(* Logix 5000 project; controller BreakGroup_US vendor 1 type 14 code 211 rev 32.16; software revision 32.05; part 6 of 8 *)
(* tags used below, declared in another part *)
   Emg_Stop : BOOL;
   HMI_ACK : BOOL;
   HMI_MAN_STN_120_STOP : BOOL;
   HMI_MAN_STN_30_STOP : BOOL;
   HMI_MAN_STN_40_STOP : BOOL;
   HMI_STN30_GRI_SETPOINT : REAL;
   HMI_STN30_HORIZ_MOVE_SETPOINT : REAL;
   HMI_STN30_VER_LIFTUP_SETPOINT : REAL;
   HMI_STN30_VER_PICK_SETPOINT : REAL;
   HMI_STN40_GRI_GRIP_POINT : REAL;
   HMI_STN40_GRI_SETPOINT : REAL;
   HMI_STN40_HORIZ_MOVE_SETPOINT : REAL;
   HMI_STN40_VER_LIFTUP_SETPOINT : REAL;
   HMI_STN40_VER_PICK_LIFTUP_SETPOINT : REAL;
   HMI_STN40_VER_PICK_SETPOINT : REAL;
   HMI_STN40_VER_PLACE_SETPOINT : REAL;
   MAN_STN_120_HOME : TIMER;
   MAN_STN_30_HOME : TIMER;
   MAN_STN_40_HOME : TIMER;
   MCP_GY_01_Gripper : MCP_Servo_01;
   MCP_GY_01_Horizontal : MCP_Servo_02;
   MCP_GY_01_Vertical : MCP_Servo_02;
   MCP_ST_30_Turntable_Motor : MCP_Servo_02;
   MCP_ST_40_Turntable_Motor : MCP_Servo_02;
   RCP_ST_120_Turntable_Motor : RCP_Servo_02;
   ST10_Trolley1Lock_Cyl_01_Extended : ALIAS FOR MCP_PT01:1:I.0;
   ST_120_Start : BOOL;
   ST_30_Start : BOOL;
   ST_40_Start : BOOL;
   STN_120_Connection_fault : BOOL;
   STN_120_Conveyor : INDEX_Block;
   STN_120_HMI_PB : SINT[2];
   STN_30_Auto_ENable : BOOL;
   STN_30_HMI_PB : SINT;
   STN_30_PRE_COND_OK : BOOL;
   STN_30_SEQ : DINT;
   STN_30_SEQUENCE_AUTO : SINT;
   STN_40_HMI_PB : SINT;
   STN_40_PRE_COND_OK : BOOL;
   STN_40_SEQ : DINT;
   STN_40_SEQUENCE_AUTO : SINT;
   T10_01 : TIMER;
   T11_01 : TIMER;
   T1_01 : TIMER;
   T2_01 : TIMER;
   T3_01 : TIMER;
   T4_01 : TIMER;
   T5_01 : TIMER;
   T6_01 : TIMER;
   T7_01 : TIMER;
   T8_01 : TIMER;
   T9_01 : TIMER;
   Test_COND_OK : DINT;
(* Station_120, continued *)

ROUTINE Manual   (* ladder *)
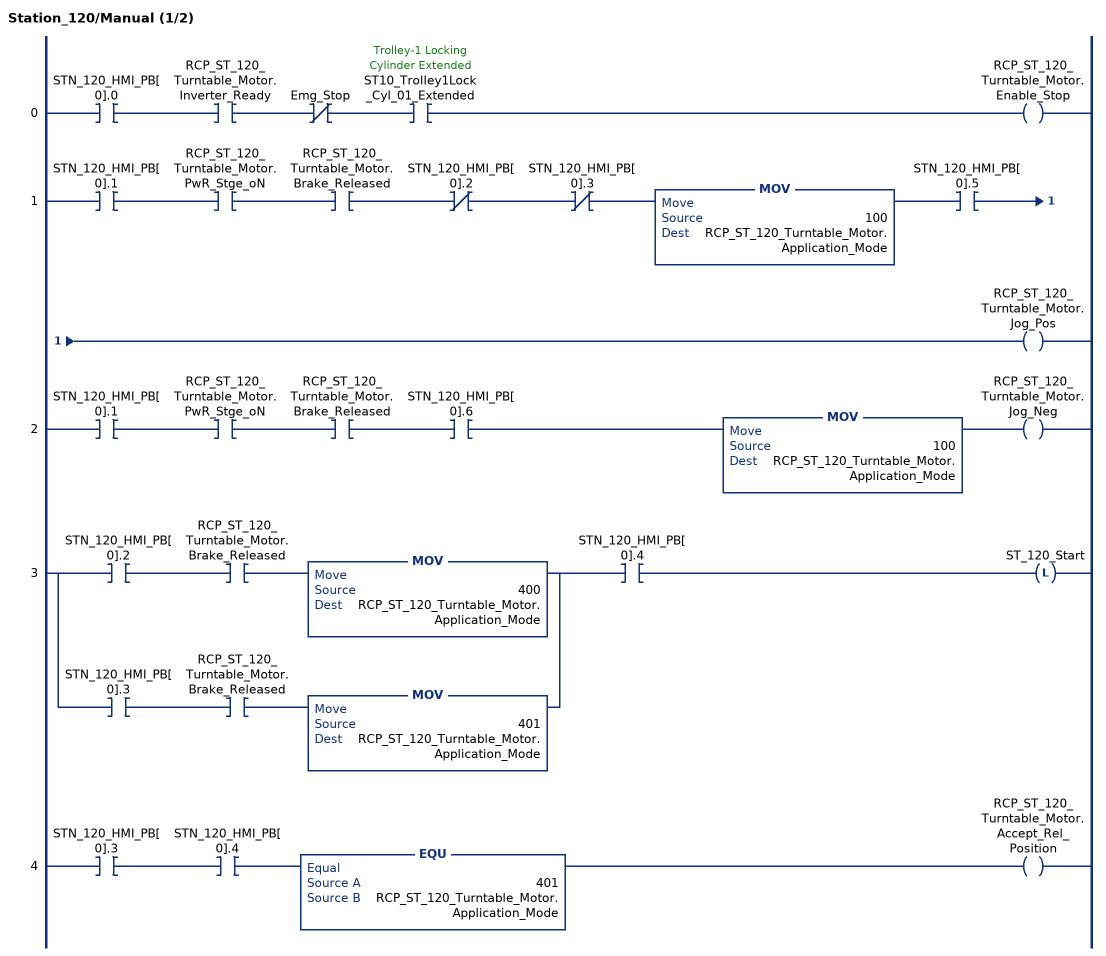
   0: XIC(STN_120_HMI_PB[0].0)XIC(RCP_ST_120_Turntable_Motor.Inverter_Ready)XIO(Emg_Stop)XIC(ST10_Trolley1Lock_Cyl_01_Extended)OTE(RCP_ST_120_Turntable_Motor.Enable_Stop);
   1: XIC(STN_120_HMI_PB[0].1)XIC(RCP_ST_120_Turntable_Motor.PwR_Stge_oN)XIC(RCP_ST_120_Turntable_Motor.Brake_Released)XIO(STN_120_HMI_PB[0].2)XIO(STN_120_HMI_PB[0].3)MOV(100,RCP_ST_120_Turntable_Motor.Application_Mode)XIC(STN_120_HMI_PB[0].5)OTE(RCP_ST_120_Turntable_Motor.Jog_Pos);
   2: XIC(STN_120_HMI_PB[0].1)XIC(RCP_ST_120_Turntable_Motor.PwR_Stge_oN)XIC(RCP_ST_120_Turntable_Motor.Brake_Released)XIC(STN_120_HMI_PB[0].6)MOV(100,RCP_ST_120_Turntable_Motor.Application_Mode)OTE(RCP_ST_120_Turntable_Motor.Jog_Neg);
   3: [XIC(STN_120_HMI_PB[0].2) XIC(RCP_ST_120_Turntable_Motor.Brake_Released) MOV(400,RCP_ST_120_Turntable_Motor.Application_Mode) ,XIC(STN_120_HMI_PB[0].3) XIC(RCP_ST_120_Turntable_Motor.Brake_Released) MOV(401,RCP_ST_120_Turntable_Motor.Application_Mode) ]XIC(STN_120_HMI_PB[0].4)OTL(ST_120_Start);
   4: XIC(STN_120_HMI_PB[0].3)XIC(STN_120_HMI_PB[0].4)EQU(401,RCP_ST_120_Turntable_Motor.Application_Mode)OTE(RCP_ST_120_Turntable_Motor.Accept_Rel_Position);
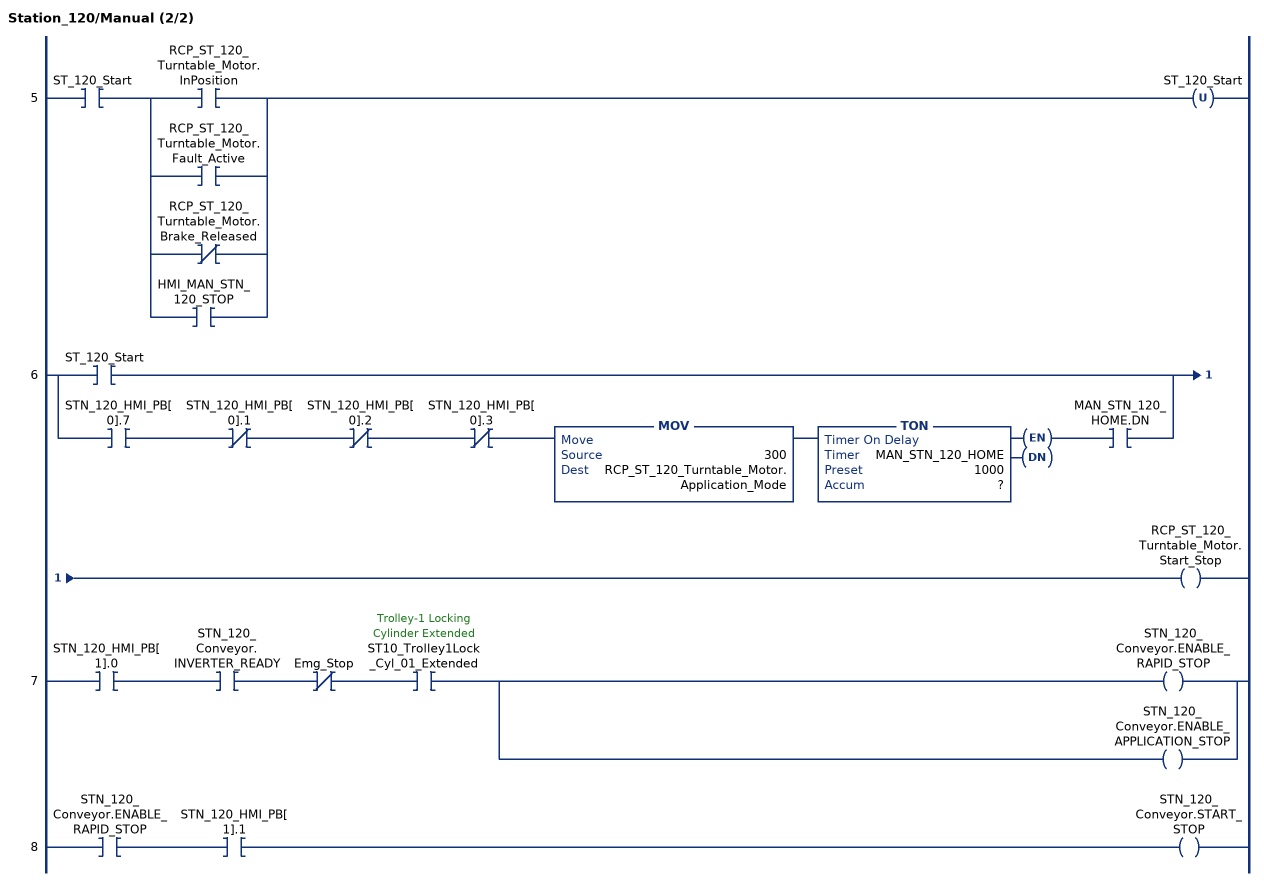
   5: XIC(ST_120_Start)[XIC(RCP_ST_120_Turntable_Motor.InPosition) ,[XIC(RCP_ST_120_Turntable_Motor.Fault_Active) ,[XIO(RCP_ST_120_Turntable_Motor.Brake_Released) ,XIC(HMI_MAN_STN_120_STOP) ] ] ]OTU(ST_120_Start);
   6: [XIC(ST_120_Start) ,XIC(STN_120_HMI_PB[0].7) XIO(STN_120_HMI_PB[0].1) XIO(STN_120_HMI_PB[0].2) XIO(STN_120_HMI_PB[0].3) MOV(300,RCP_ST_120_Turntable_Motor.Application_Mode) TON(MAN_STN_120_HOME,?,?) XIC(MAN_STN_120_HOME.DN) ]OTE(RCP_ST_120_Turntable_Motor.Start_Stop);
   7: XIC(STN_120_HMI_PB[1].0)XIC(STN_120_Conveyor.INVERTER_READY)XIO(Emg_Stop)XIC(ST10_Trolley1Lock_Cyl_01_Extended)[OTE(STN_120_Conveyor.ENABLE_RAPID_STOP) ,OTE(STN_120_Conveyor.ENABLE_APPLICATION_STOP) ];
   8: XIC(STN_120_Conveyor.ENABLE_RAPID_STOP)XIC(STN_120_HMI_PB[1].1)OTE(STN_120_Conveyor.START_STOP);
END_ROUTINE

ROUTINE Servo   (* ladder *)
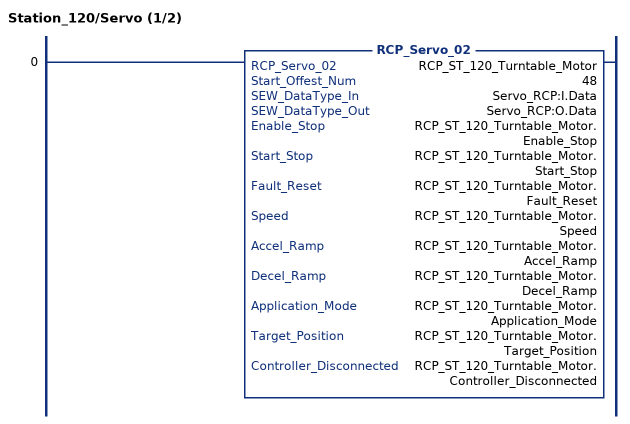
   0: RCP_Servo_02(RCP_ST_120_Turntable_Motor,48,Servo_RCP:I.Data,Servo_RCP:O.Data,RCP_ST_120_Turntable_Motor.Enable_Stop,RCP_ST_120_Turntable_Motor.Start_Stop,RCP_ST_120_Turntable_Motor.Fault_Reset,RCP_ST_120_Turntable_Motor.Speed,RCP_ST_120_Turntable_Motor.Accel_Ramp,RCP_ST_120_Turntable_Motor.Decel_Ramp,RCP_ST_120_Turntable_Motor.Application_Mode,RCP_ST_120_Turntable_Motor.Target_Position,RCP_ST_120_Turntable_Motor.Controller_Disconnected);
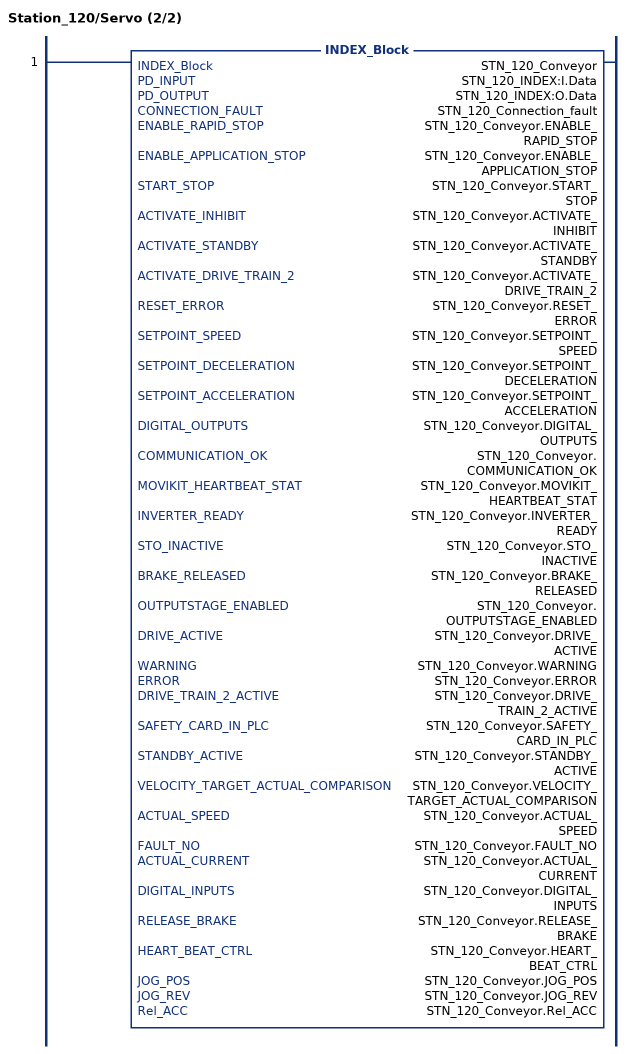
   1: INDEX_Block(STN_120_Conveyor,STN_120_INDEX:I.Data,STN_120_INDEX:O.Data,STN_120_Connection_fault,STN_120_Conveyor.ENABLE_RAPID_STOP,STN_120_Conveyor.ENABLE_APPLICATION_STOP,STN_120_Conveyor.START_STOP,STN_120_Conveyor.ACTIVATE_INHIBIT,STN_120_Conveyor.ACTIVATE_STANDBY,STN_120_Conveyor.ACTIVATE_DRIVE_TRAIN_2,STN_120_Conveyor.RESET_ERROR,STN_120_Conveyor.SETPOINT_SPEED,STN_120_Conveyor.SETPOINT_DECELERATION,STN_120_Conveyor.SETPOINT_ACCELERATION,STN_120_Conveyor.DIGITAL_OUTPUTS,STN_120_Conveyor.COMMUNICATION_OK,STN_120_Conveyor.MOVIKIT_HEARTBEAT_STAT,STN_120_Conveyor.INVERTER_READY,STN_120_Conveyor.STO_INACTIVE,STN_120_Conveyor.BRAKE_RELEASED,STN_120_Conveyor.OUTPUTSTAGE_ENABLED,STN_120_Conveyor.DRIVE_ACTIVE,STN_120_Conveyor.WARNING,STN_120_Conveyor.ERROR,STN_120_Conveyor.DRIVE_TRAIN_2_ACTIVE,STN_120_Conveyor.SAFETY_CARD_IN_PLC,STN_120_Conveyor.STANDBY_ACTIVE,STN_120_Conveyor.VELOCITY_TARGET_ACTUAL_COMPARISON,STN_120_Conveyor.ACTUAL_SPEED,STN_120_Conveyor.FAULT_NO,STN_120_Conveyor.ACTUAL_CURRENT,STN_120_Conveyor.DIGITAL_INPUTS,STN_120_Conveyor.RELEASE_BRAKE,STN_120_Conveyor.HEART_BEAT_CTRL,STN_120_Conveyor.JOG_POS,STN_120_Conveyor.JOG_REV,STN_120_Conveyor.Rel_ACC);
END_ROUTINE
END_PROGRAM

PROGRAM Station_20
END_PROGRAM

PROGRAM Station_30   (* main routine Main *)

ROUTINE Main   (* ladder *)
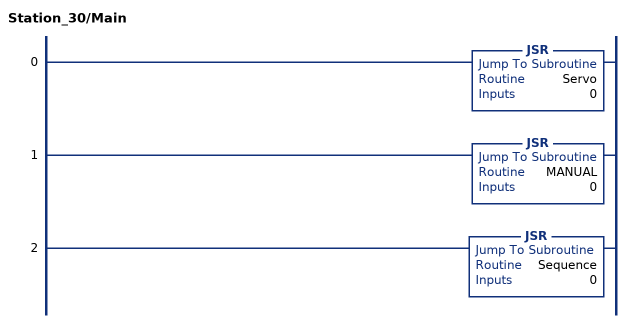
   0: JSR(Servo,0);
   1: JSR(MANUAL,0);
   2: JSR(Sequence,0);
END_ROUTINE

ROUTINE MANUAL   (* ladder *)
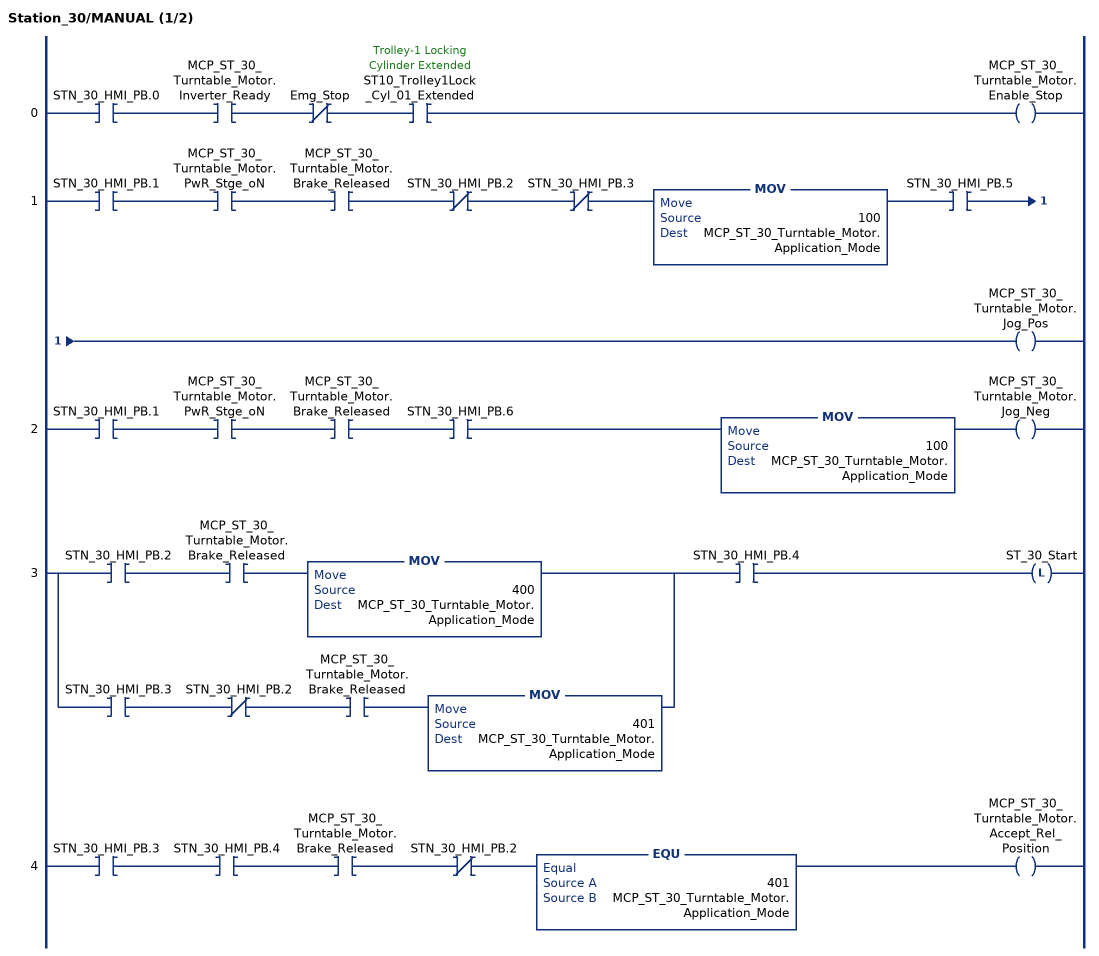
   0: XIC(STN_30_HMI_PB.0)XIC(MCP_ST_30_Turntable_Motor.Inverter_Ready)XIO(Emg_Stop)XIC(ST10_Trolley1Lock_Cyl_01_Extended)OTE(MCP_ST_30_Turntable_Motor.Enable_Stop);
   1: XIC(STN_30_HMI_PB.1)XIC(MCP_ST_30_Turntable_Motor.PwR_Stge_oN)XIC(MCP_ST_30_Turntable_Motor.Brake_Released)XIO(STN_30_HMI_PB.2)XIO(STN_30_HMI_PB.3)MOV(100,MCP_ST_30_Turntable_Motor.Application_Mode)XIC(STN_30_HMI_PB.5)OTE(MCP_ST_30_Turntable_Motor.Jog_Pos);
   2: XIC(STN_30_HMI_PB.1)XIC(MCP_ST_30_Turntable_Motor.PwR_Stge_oN)XIC(MCP_ST_30_Turntable_Motor.Brake_Released)XIC(STN_30_HMI_PB.6)MOV(100,MCP_ST_30_Turntable_Motor.Application_Mode)OTE(MCP_ST_30_Turntable_Motor.Jog_Neg);
   3: [XIC(STN_30_HMI_PB.2) XIC(MCP_ST_30_Turntable_Motor.Brake_Released) MOV(400,MCP_ST_30_Turntable_Motor.Application_Mode) ,XIC(STN_30_HMI_PB.3) XIO(STN_30_HMI_PB.2) XIC(MCP_ST_30_Turntable_Motor.Brake_Released) MOV(401,MCP_ST_30_Turntable_Motor.Application_Mode) ]XIC(STN_30_HMI_PB.4)OTL(ST_30_Start);
   4: XIC(STN_30_HMI_PB.3)XIC(STN_30_HMI_PB.4)XIC(MCP_ST_30_Turntable_Motor.Brake_Released)XIO(STN_30_HMI_PB.2)EQU(401,MCP_ST_30_Turntable_Motor.Application_Mode)OTE(MCP_ST_30_Turntable_Motor.Accept_Rel_Position);
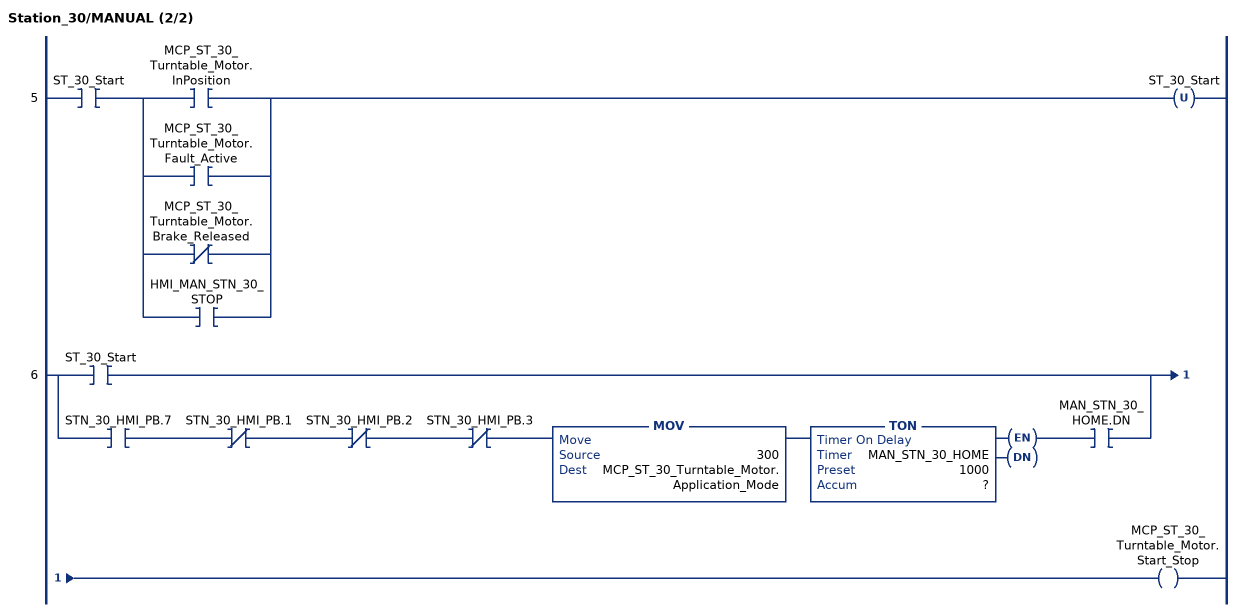
   5: XIC(ST_30_Start)[XIC(MCP_ST_30_Turntable_Motor.InPosition) ,[XIC(MCP_ST_30_Turntable_Motor.Fault_Active) ,[XIO(MCP_ST_30_Turntable_Motor.Brake_Released) ,XIC(HMI_MAN_STN_30_STOP) ] ] ]OTU(ST_30_Start);
   6: [XIC(ST_30_Start) ,XIC(STN_30_HMI_PB.7) XIO(STN_30_HMI_PB.1) XIO(STN_30_HMI_PB.2) XIO(STN_30_HMI_PB.3) MOV(300,MCP_ST_30_Turntable_Motor.Application_Mode) TON(MAN_STN_30_HOME,?,?) XIC(MAN_STN_30_HOME.DN) ]OTE(MCP_ST_30_Turntable_Motor.Start_Stop);
END_ROUTINE

ROUTINE Sequence   (* ladder *)
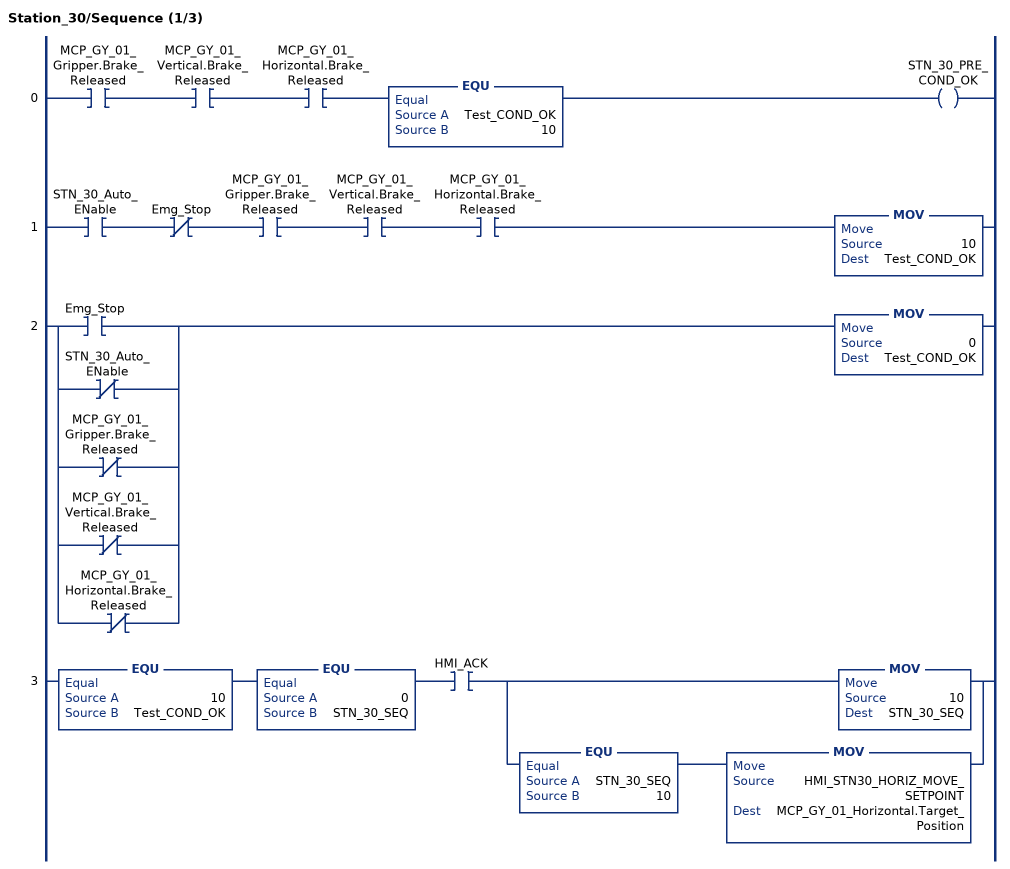
   0: XIC(MCP_GY_01_Gripper.Brake_Released)XIC(MCP_GY_01_Vertical.Brake_Released)XIC(MCP_GY_01_Horizontal.Brake_Released)EQU(Test_COND_OK,10)OTE(STN_30_PRE_COND_OK);
   1: XIC(STN_30_Auto_ENable)XIO(Emg_Stop)XIC(MCP_GY_01_Gripper.Brake_Released)XIC(MCP_GY_01_Vertical.Brake_Released)XIC(MCP_GY_01_Horizontal.Brake_Released)MOV(10,Test_COND_OK);
   2: [XIC(Emg_Stop) ,[XIO(STN_30_Auto_ENable) ,[XIO(MCP_GY_01_Gripper.Brake_Released) ,[XIO(MCP_GY_01_Vertical.Brake_Released) ,XIO(MCP_GY_01_Horizontal.Brake_Released) ] ] ] ]MOV(0,Test_COND_OK);
   3: EQU(10,Test_COND_OK)EQU(0,STN_30_SEQ)XIC(HMI_ACK)[MOV(10,STN_30_SEQ) ,EQU(STN_30_SEQ,10) MOV(HMI_STN30_HORIZ_MOVE_SETPOINT,MCP_GY_01_Horizontal.Target_Position) ];
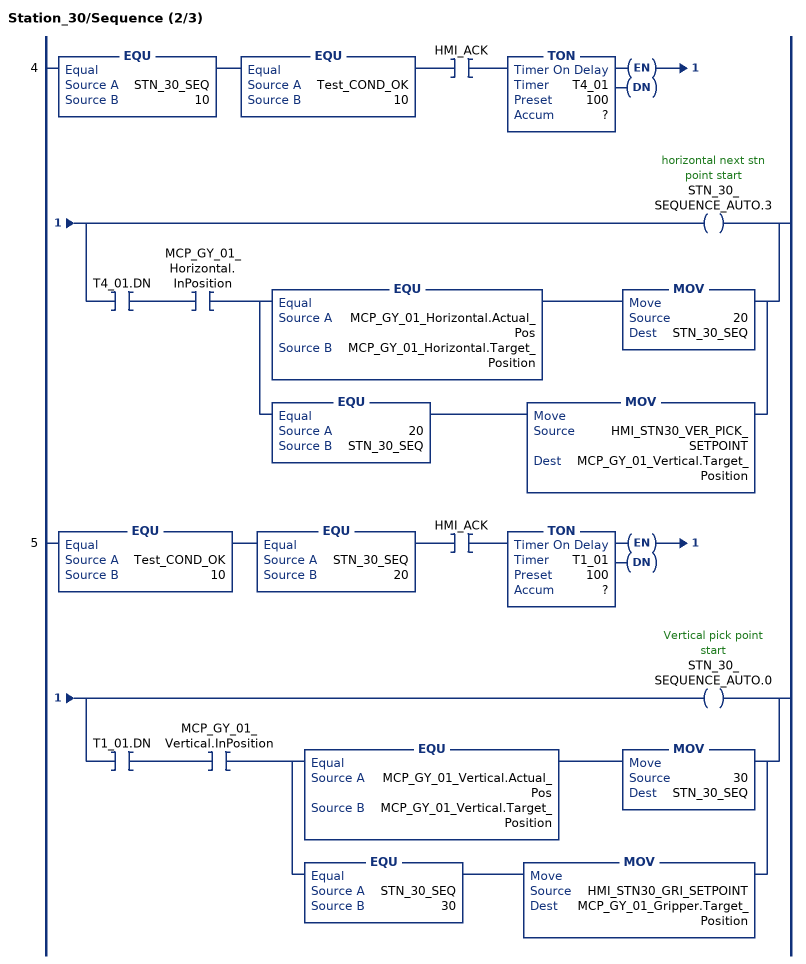
   4: EQU(STN_30_SEQ,10)EQU(Test_COND_OK,10)XIC(HMI_ACK)TON(T4_01,?,?)[OTE(STN_30_SEQUENCE_AUTO.3) ,XIC(T4_01.DN) XIC(MCP_GY_01_Horizontal.InPosition) [EQU(MCP_GY_01_Horizontal.Actual_Pos,MCP_GY_01_Horizontal.Target_Position) MOV(20,STN_30_SEQ) ,EQU(20,STN_30_SEQ) MOV(HMI_STN30_VER_PICK_SETPOINT,MCP_GY_01_Vertical.Target_Position) ] ];
   5: EQU(Test_COND_OK,10)EQU(STN_30_SEQ,20)XIC(HMI_ACK)TON(T1_01,?,?)[OTE(STN_30_SEQUENCE_AUTO.0) ,XIC(T1_01.DN) XIC(MCP_GY_01_Vertical.InPosition) [EQU(MCP_GY_01_Vertical.Actual_Pos,MCP_GY_01_Vertical.Target_Position) MOV(30,STN_30_SEQ) ,EQU(STN_30_SEQ,30) MOV(HMI_STN30_GRI_SETPOINT,MCP_GY_01_Gripper.Target_Position) ] ];
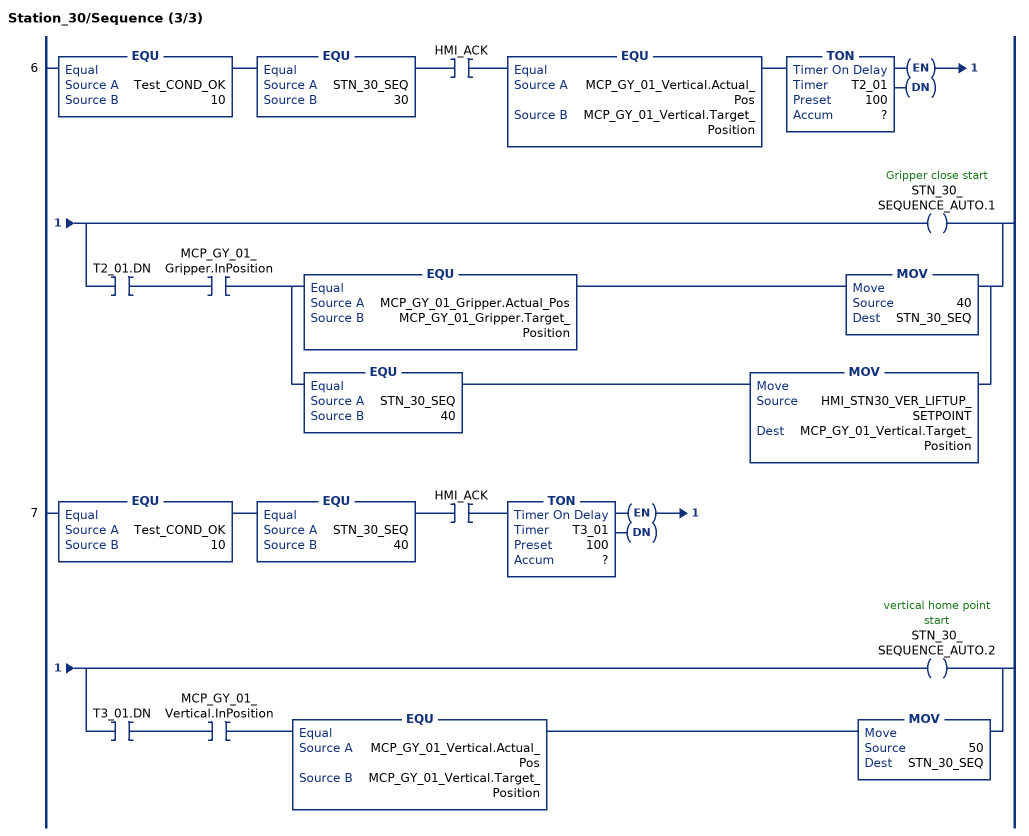
   6: EQU(Test_COND_OK,10)EQU(STN_30_SEQ,30)XIC(HMI_ACK)EQU(MCP_GY_01_Vertical.Actual_Pos,MCP_GY_01_Vertical.Target_Position)TON(T2_01,?,?)[OTE(STN_30_SEQUENCE_AUTO.1) ,XIC(T2_01.DN) XIC(MCP_GY_01_Gripper.InPosition) [EQU(MCP_GY_01_Gripper.Actual_Pos,MCP_GY_01_Gripper.Target_Position) MOV(40,STN_30_SEQ) ,EQU(STN_30_SEQ,40) MOV(HMI_STN30_VER_LIFTUP_SETPOINT,MCP_GY_01_Vertical.Target_Position) ] ];
   7: EQU(Test_COND_OK,10)EQU(STN_30_SEQ,40)XIC(HMI_ACK)TON(T3_01,?,?)[OTE(STN_30_SEQUENCE_AUTO.2) ,XIC(T3_01.DN) XIC(MCP_GY_01_Vertical.InPosition) EQU(MCP_GY_01_Vertical.Actual_Pos,MCP_GY_01_Vertical.Target_Position) MOV(50,STN_30_SEQ) ];
END_ROUTINE

ROUTINE Servo   (* ladder *)
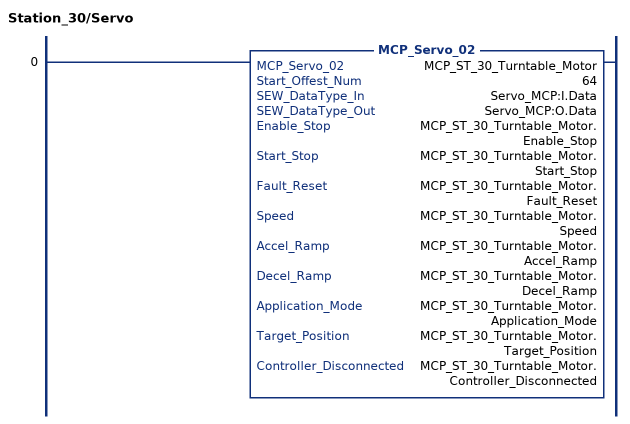
   0: MCP_Servo_02(MCP_ST_30_Turntable_Motor,64,Servo_MCP:I.Data,Servo_MCP:O.Data,MCP_ST_30_Turntable_Motor.Enable_Stop,MCP_ST_30_Turntable_Motor.Start_Stop,MCP_ST_30_Turntable_Motor.Fault_Reset,MCP_ST_30_Turntable_Motor.Speed,MCP_ST_30_Turntable_Motor.Accel_Ramp,MCP_ST_30_Turntable_Motor.Decel_Ramp,MCP_ST_30_Turntable_Motor.Application_Mode,MCP_ST_30_Turntable_Motor.Target_Position,MCP_ST_30_Turntable_Motor.Controller_Disconnected);
END_ROUTINE
END_PROGRAM

PROGRAM Station_40   (* main routine Main *)

ROUTINE Main   (* ladder *)
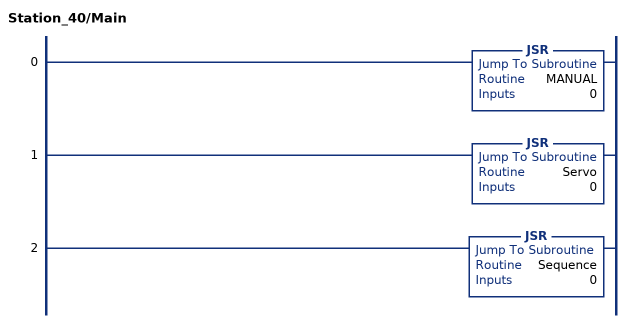
   0: JSR(MANUAL,0);
   1: JSR(Servo,0);
   2: JSR(Sequence,0);
END_ROUTINE

ROUTINE MANUAL   (* ladder *)
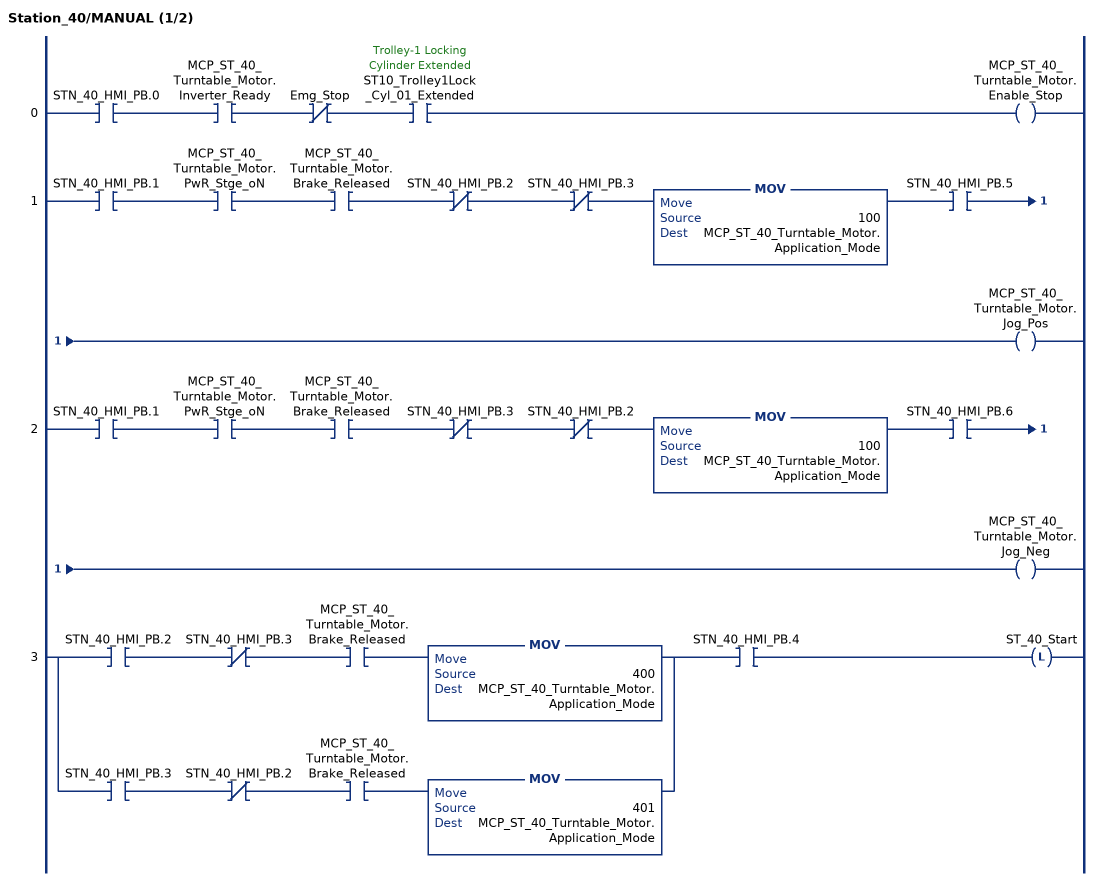
   0: XIC(STN_40_HMI_PB.0)XIC(MCP_ST_40_Turntable_Motor.Inverter_Ready)XIO(Emg_Stop)XIC(ST10_Trolley1Lock_Cyl_01_Extended)OTE(MCP_ST_40_Turntable_Motor.Enable_Stop);
   1: XIC(STN_40_HMI_PB.1)XIC(MCP_ST_40_Turntable_Motor.PwR_Stge_oN)XIC(MCP_ST_40_Turntable_Motor.Brake_Released)XIO(STN_40_HMI_PB.2)XIO(STN_40_HMI_PB.3)MOV(100,MCP_ST_40_Turntable_Motor.Application_Mode)XIC(STN_40_HMI_PB.5)OTE(MCP_ST_40_Turntable_Motor.Jog_Pos);
   2: XIC(STN_40_HMI_PB.1)XIC(MCP_ST_40_Turntable_Motor.PwR_Stge_oN)XIC(MCP_ST_40_Turntable_Motor.Brake_Released)XIO(STN_40_HMI_PB.3)XIO(STN_40_HMI_PB.2)MOV(100,MCP_ST_40_Turntable_Motor.Application_Mode)XIC(STN_40_HMI_PB.6)OTE(MCP_ST_40_Turntable_Motor.Jog_Neg);
   3: [XIC(STN_40_HMI_PB.2) XIO(STN_40_HMI_PB.3) XIC(MCP_ST_40_Turntable_Motor.Brake_Released) MOV(400,MCP_ST_40_Turntable_Motor.Application_Mode) ,XIC(STN_40_HMI_PB.3) XIO(STN_40_HMI_PB.2) XIC(MCP_ST_40_Turntable_Motor.Brake_Released) MOV(401,MCP_ST_40_Turntable_Motor.Application_Mode) ]XIC(STN_40_HMI_PB.4)OTL(ST_40_Start);
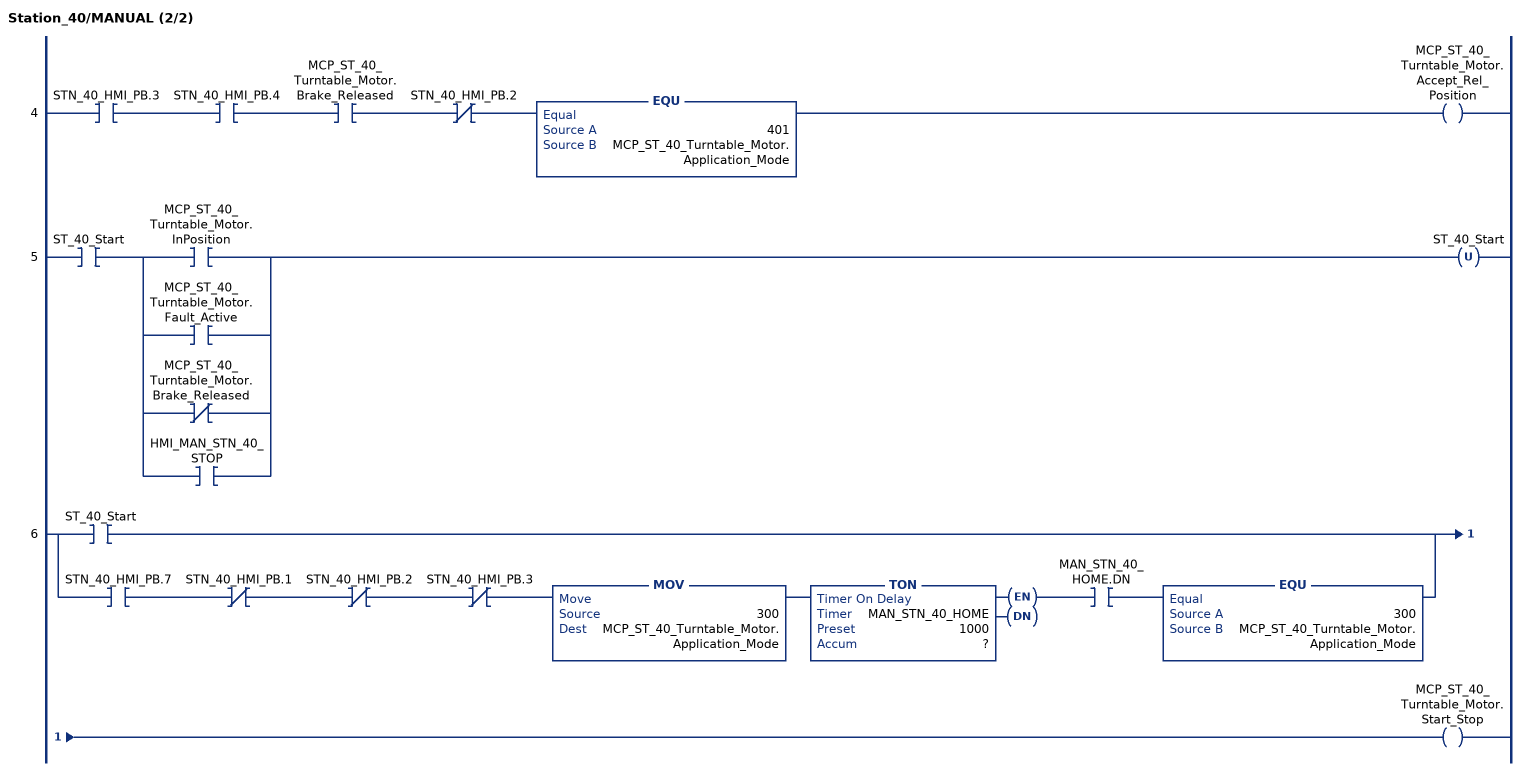
   4: XIC(STN_40_HMI_PB.3)XIC(STN_40_HMI_PB.4)XIC(MCP_ST_40_Turntable_Motor.Brake_Released)XIO(STN_40_HMI_PB.2)EQU(401,MCP_ST_40_Turntable_Motor.Application_Mode)OTE(MCP_ST_40_Turntable_Motor.Accept_Rel_Position);
   5: XIC(ST_40_Start)[XIC(MCP_ST_40_Turntable_Motor.InPosition) ,[XIC(MCP_ST_40_Turntable_Motor.Fault_Active) ,[XIO(MCP_ST_40_Turntable_Motor.Brake_Released) ,XIC(HMI_MAN_STN_40_STOP) ] ] ]OTU(ST_40_Start);
   6: [XIC(ST_40_Start) ,XIC(STN_40_HMI_PB.7) XIO(STN_40_HMI_PB.1) XIO(STN_40_HMI_PB.2) XIO(STN_40_HMI_PB.3) MOV(300,MCP_ST_40_Turntable_Motor.Application_Mode) TON(MAN_STN_40_HOME,?,?) XIC(MAN_STN_40_HOME.DN) EQU(300,MCP_ST_40_Turntable_Motor.Application_Mode) ]OTE(MCP_ST_40_Turntable_Motor.Start_Stop);
END_ROUTINE

ROUTINE Sequence   (* ladder *)
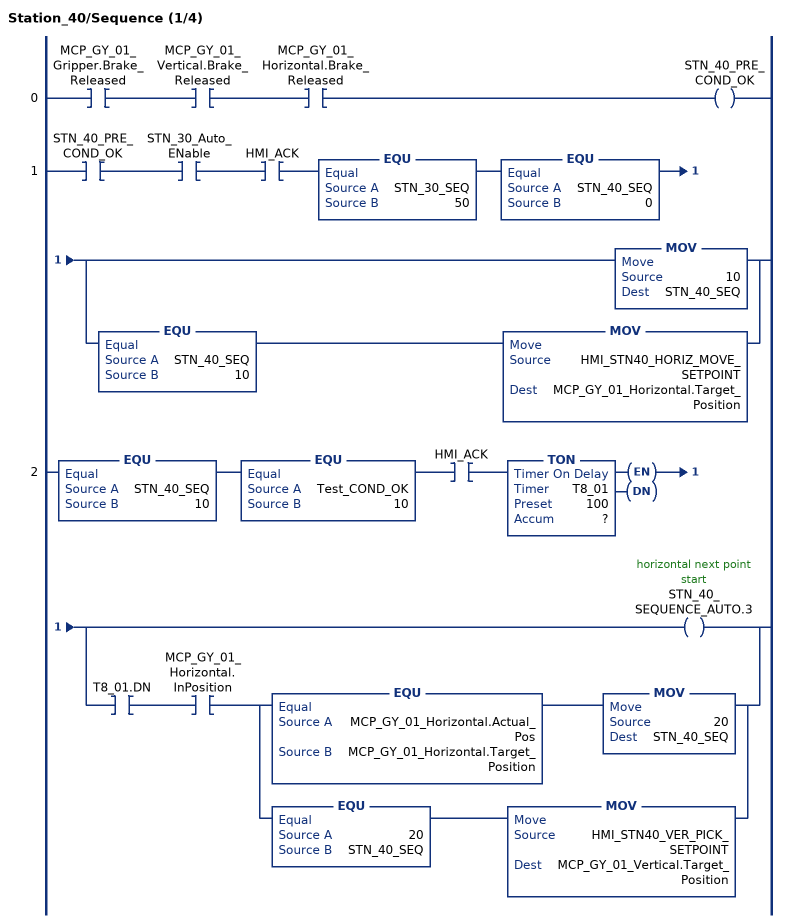
   0: XIC(MCP_GY_01_Gripper.Brake_Released)XIC(MCP_GY_01_Vertical.Brake_Released)XIC(MCP_GY_01_Horizontal.Brake_Released)OTE(STN_40_PRE_COND_OK);
   1: XIC(STN_40_PRE_COND_OK)XIC(STN_30_Auto_ENable)XIC(HMI_ACK)EQU(STN_30_SEQ,50)EQU(STN_40_SEQ,0)[MOV(10,STN_40_SEQ) ,EQU(STN_40_SEQ,10) MOV(HMI_STN40_HORIZ_MOVE_SETPOINT,MCP_GY_01_Horizontal.Target_Position) ];
   2: EQU(STN_40_SEQ,10)EQU(Test_COND_OK,10)XIC(HMI_ACK)TON(T8_01,?,?)[OTE(STN_40_SEQUENCE_AUTO.3) ,XIC(T8_01.DN) XIC(MCP_GY_01_Horizontal.InPosition) [EQU(MCP_GY_01_Horizontal.Actual_Pos,MCP_GY_01_Horizontal.Target_Position) MOV(20,STN_40_SEQ) ,EQU(20,STN_40_SEQ) MOV(HMI_STN40_VER_PICK_SETPOINT,MCP_GY_01_Vertical.Target_Position) ] ];
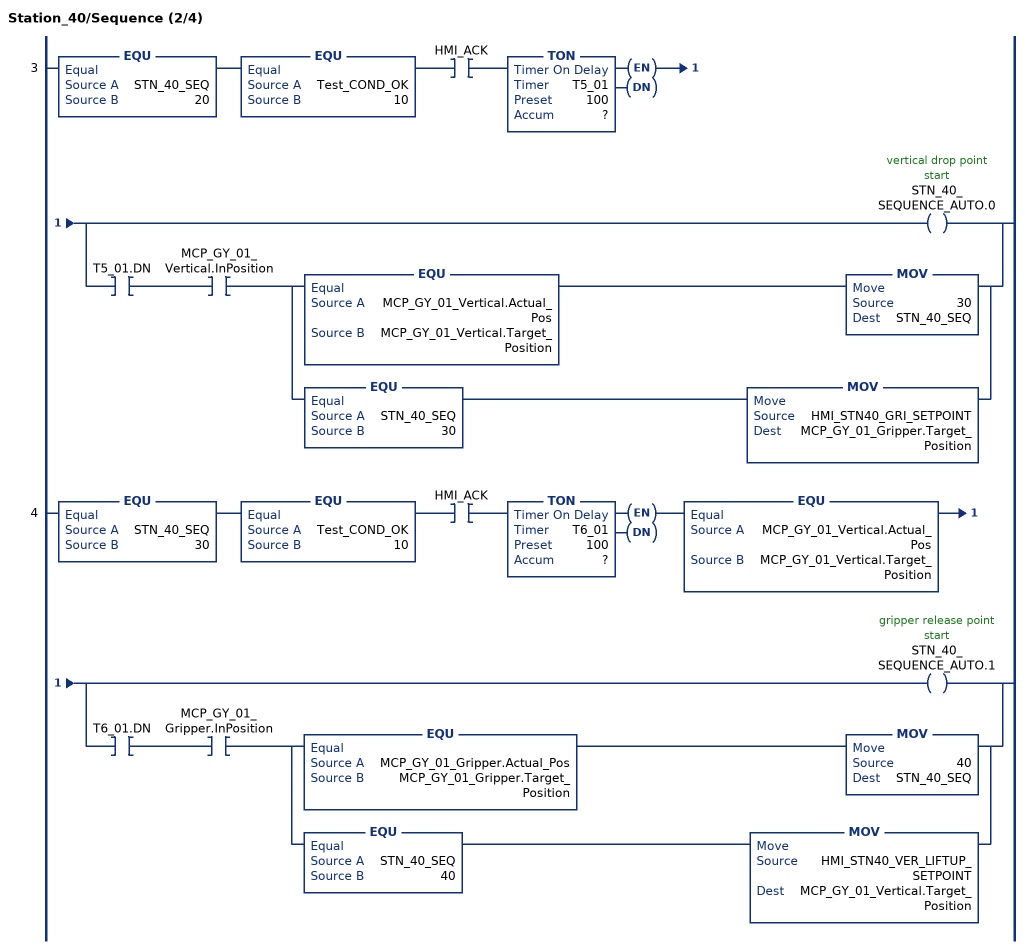
   3: EQU(STN_40_SEQ,20)EQU(Test_COND_OK,10)XIC(HMI_ACK)TON(T5_01,?,?)[OTE(STN_40_SEQUENCE_AUTO.0) ,XIC(T5_01.DN) XIC(MCP_GY_01_Vertical.InPosition) [EQU(MCP_GY_01_Vertical.Actual_Pos,MCP_GY_01_Vertical.Target_Position) MOV(30,STN_40_SEQ) ,EQU(STN_40_SEQ,30) MOV(HMI_STN40_GRI_SETPOINT,MCP_GY_01_Gripper.Target_Position) ] ];
   4: EQU(STN_40_SEQ,30)EQU(Test_COND_OK,10)XIC(HMI_ACK)TON(T6_01,?,?)EQU(MCP_GY_01_Vertical.Actual_Pos,MCP_GY_01_Vertical.Target_Position)[OTE(STN_40_SEQUENCE_AUTO.1) ,XIC(T6_01.DN) XIC(MCP_GY_01_Gripper.InPosition) [EQU(MCP_GY_01_Gripper.Actual_Pos,MCP_GY_01_Gripper.Target_Position) MOV(40,STN_40_SEQ) ,EQU(STN_40_SEQ,40) MOV(HMI_STN40_VER_LIFTUP_SETPOINT,MCP_GY_01_Vertical.Target_Position) ] ];
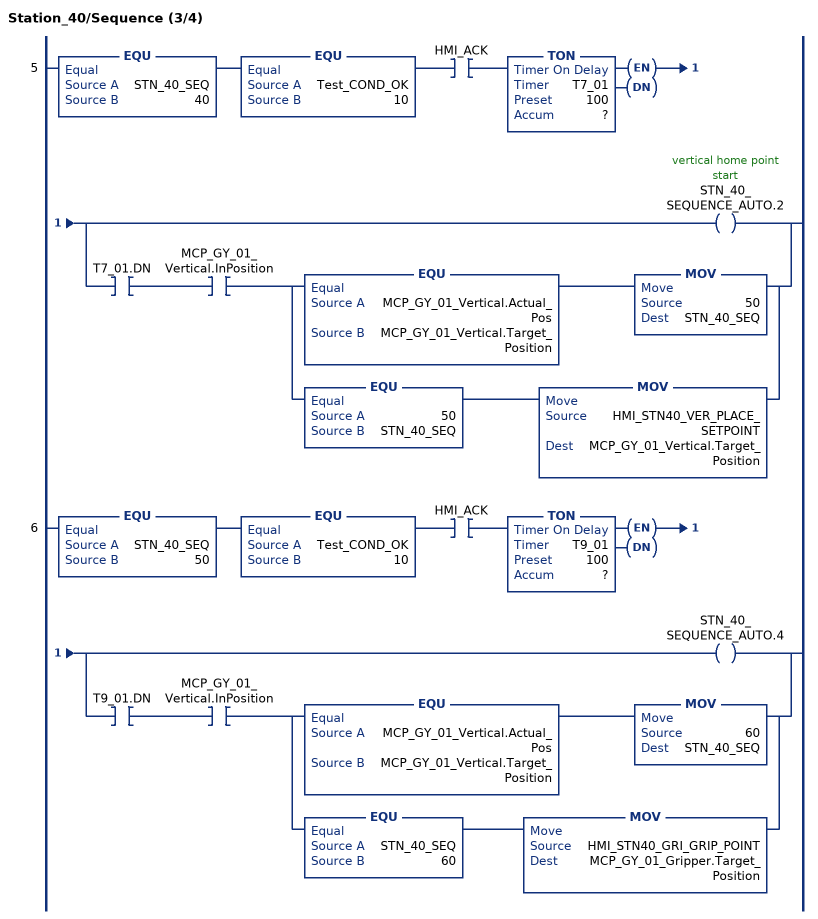
   5: EQU(STN_40_SEQ,40)EQU(Test_COND_OK,10)XIC(HMI_ACK)TON(T7_01,?,?)[OTE(STN_40_SEQUENCE_AUTO.2) ,XIC(T7_01.DN) XIC(MCP_GY_01_Vertical.InPosition) [EQU(MCP_GY_01_Vertical.Actual_Pos,MCP_GY_01_Vertical.Target_Position) MOV(50,STN_40_SEQ) ,EQU(50,STN_40_SEQ) MOV(HMI_STN40_VER_PLACE_SETPOINT,MCP_GY_01_Vertical.Target_Position) ] ];
   6: EQU(STN_40_SEQ,50)EQU(Test_COND_OK,10)XIC(HMI_ACK)TON(T9_01,?,?)[OTE(STN_40_SEQUENCE_AUTO.4) ,XIC(T9_01.DN) XIC(MCP_GY_01_Vertical.InPosition) [EQU(MCP_GY_01_Vertical.Actual_Pos,MCP_GY_01_Vertical.Target_Position) MOV(60,STN_40_SEQ) ,EQU(STN_40_SEQ,60) MOV(HMI_STN40_GRI_GRIP_POINT,MCP_GY_01_Gripper.Target_Position) ] ];
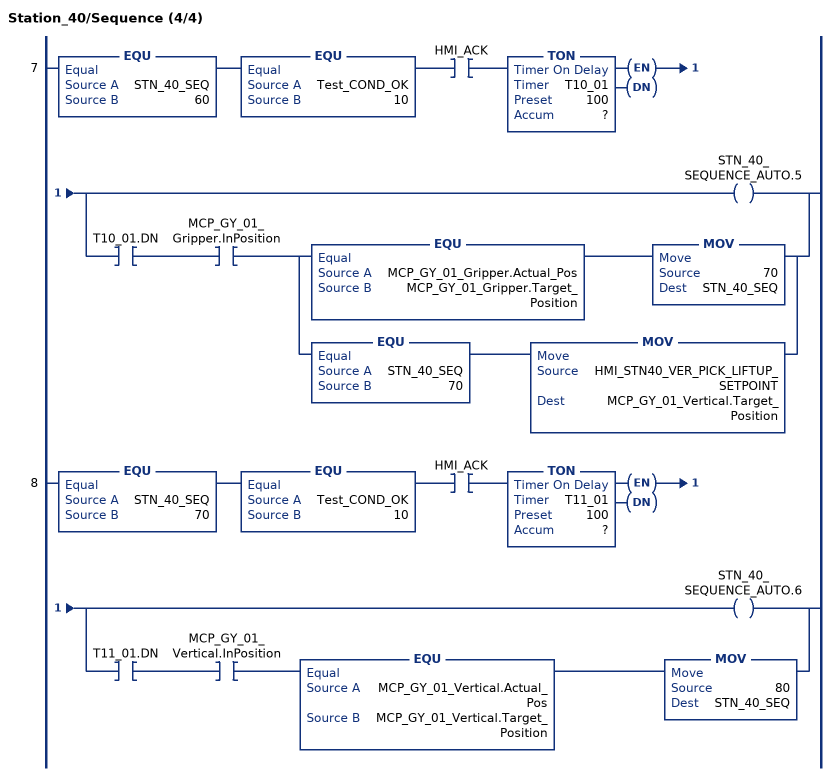
   7: EQU(STN_40_SEQ,60)EQU(Test_COND_OK,10)XIC(HMI_ACK)TON(T10_01,?,?)[OTE(STN_40_SEQUENCE_AUTO.5) ,XIC(T10_01.DN) XIC(MCP_GY_01_Gripper.InPosition) [EQU(MCP_GY_01_Gripper.Actual_Pos,MCP_GY_01_Gripper.Target_Position) MOV(70,STN_40_SEQ) ,EQU(STN_40_SEQ,70) MOV(HMI_STN40_VER_PICK_LIFTUP_SETPOINT,MCP_GY_01_Vertical.Target_Position) ] ];
   8: EQU(STN_40_SEQ,70)EQU(Test_COND_OK,10)XIC(HMI_ACK)TON(T11_01,?,?)[OTE(STN_40_SEQUENCE_AUTO.6) ,XIC(T11_01.DN) XIC(MCP_GY_01_Vertical.InPosition) EQU(MCP_GY_01_Vertical.Actual_Pos,MCP_GY_01_Vertical.Target_Position) MOV(80,STN_40_SEQ) ];
END_ROUTINE
